(* PLC project Untitled1, Beckhoff Automation GmbH TwinCAT PLC Control 3.5.13.20 *)
(* stored: creationDateTime 2021-03-30T13:50:39.4131495, modificationDateTime 2021-03-30T13:50:39.4171496 *)

FUNCTION_BLOCK FB_MoveVelocityAutoChange
  VAR_INPUT
    Execute : BOOL;
    Velocity : LREAL;
    Acceleration : LREAL;
    Deceleration : LREAL;
    Jerk : LREAL;
  END_VAR
  VAR_OUTPUT
    Busy : BOOL;
    Error : BOOL;
    ErrorID : UDINT;
    CommandAborted : BOOL;
  END_VAR
  VAR
    Step : INT;
    MC_MoveVelocity : MC_MoveVelocity;
    MC_MoveVelocity2 : MC_MoveVelocity;
    VelocityChanged : BOOL;
    VelocityOld : LREAL;
    TrigbExecute : R_TRIG;
    TonTimeOut : TON;
  END_VAR
  VAR_IN_OUT
    Axis : AXIS_REF;
  END_VAR

            IF Execute = TRUE THEN
	IF VelocityOld <> Velocity THEN
		VelocityChanged:=TRUE;
	END_IF
END_IF
IF Velocity < 0 THEN
	MC_MoveVelocity.Direction :=MC_Negative_Direction;
	MC_MoveVelocity2.Direction:=MC_Negative_Direction;
ELSE
	MC_MoveVelocity.Direction :=MC_Positive_Direction;
	MC_MoveVelocity2.Direction:=MC_Positive_Direction;
END_IF

MC_MoveVelocity(
	Axis:=Axis , 
	Execute:=Execute AND Step=0,
	Velocity:=ABS( Velocity),
	Acceleration:=Acceleration ,
	Deceleration:=Deceleration ,
	Jerk:=Jerk );
MC_MoveVelocity2(
	Axis:=Axis , 
	Execute:=Execute AND Step =1,
	Velocity:= ABS( Velocity),
	Acceleration:=Acceleration ,
	Deceleration:=Deceleration , 
	Jerk:=Jerk );

CASE Step OF
0:
	IF VelocityChanged THEN
		Step:=1;
		MC_MoveVelocity(
			Axis:=Axis , 
			Execute:=FALSE);
		MC_MoveVelocity2(
			Axis:=Axis , 
			Execute:=FALSE);
		VelocityChanged:=FALSE;
	END_IF
	Busy:=MC_MoveVelocity.Busy;
	Error:=MC_MoveVelocity.Error;
	ErrorID:=MC_MoveVelocity.ErrorID;
	CommandAborted:=MC_MoveVelocity.CommandAborted;

1:
	IF VelocityChanged THEN
		Step:=0;
		MC_MoveVelocity(
			Axis:=Axis , 
			Execute:=FALSE);
		MC_MoveVelocity2(
			Axis:=Axis , 
			Execute:=FALSE);
		VelocityChanged:=FALSE;
	END_IF
	Busy:=MC_MoveVelocity2.Busy;
	Error:=MC_MoveVelocity2.Error;
	ErrorID:=MC_MoveVelocity2.ErrorID;
	CommandAborted:=MC_MoveVelocity2.CommandAborted;
END_CASE

VelocityOld:=Velocity;
          
END_FUNCTION_BLOCK
